Yaskawa INFORM job: tank_top_cylinder_program.JBI

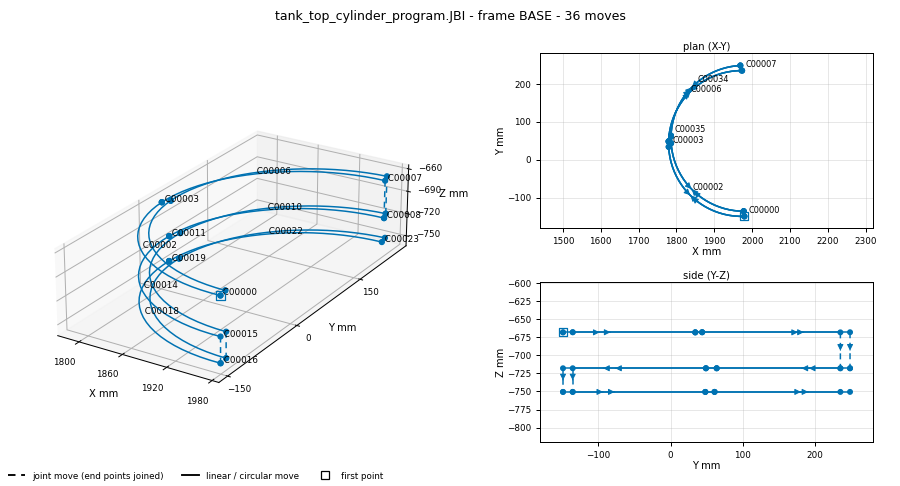
[picture p0: tool path of tank_top_cylinder_program.JBI in frame BASE, 36 of 53 moves have a stored position in this frame; points joined in program order, loops and branches not executed]
/JOB
//NAME tank_top_cylinder_program
//POS
///NPOS 48,0,48,0,0,0
///TOOL 0
///POSTYPE BASE
///RECTAN
///RCONF 0,0,0,0,0,0,0,0,0,0,0,0,0,0,0,0,0,0,0,0,0,0,0,0
C00000=1979.397693,-149.249816,-667.882960,175.000000,-60.000000,92.235388
C00001=1979.397693,-149.249816,-667.882960,175.000000,-60.000000,92.235388
C00002=1833.061579,-90.299080,-667.882960,175.000000,-60.000000,43.881048
C00003=1779.487286,34.344834,-667.882960,175.000000,-60.000000,5.000000
C00004=1779.487286,34.344834,-667.882960,175.000000,-60.000000,5.000000
C00005=1779.487286,34.344834,-667.882960,175.000000,-60.000000,5.000000
C00006=1826.412747,169.432456,-667.882960,-175.000000,-60.000000,-40.948275
C00007=1973.618558,235.799618,-667.882960,-175.000000,-60.000000,-90.515634
C00008=1973.589783,235.799875,-717.744460,175.000000,-60.000000,-90.507073
C00009=1973.589783,235.799875,-717.744460,175.000000,-60.000000,-90.507073
C00010=1835.629981,179.330426,-717.744460,175.000000,-60.000000,-44.972576
C00011=1779.374912,49.143354,-717.744460,-175.000000,-60.000000,-5.000000
C00012=1779.374912,49.143354,-717.744460,-175.000000,-60.000000,-5.000000
C00013=1779.374912,49.143354,-717.744460,-175.000000,-60.000000,-5.000000
C00014=1834.422880,-91.700324,-717.744460,-175.000000,-60.000000,44.462219
C00015=1979.256218,-149.255286,-717.744460,175.000000,-60.000000,92.193270
C00016=1979.223949,-149.256519,-750.568460,175.000000,-60.000000,92.183664
C00017=1979.223949,-149.256519,-750.568460,175.000000,-60.000000,92.183664
C00018=1835.536121,-92.825377,-750.568460,175.000000,-60.000000,44.933056
C00019=1779.350875,48.304771,-750.568460,-175.000000,-60.000000,-5.000000
C00020=1779.350875,48.304771,-750.568460,-175.000000,-60.000000,-5.000000
C00021=1779.350875,48.304771,-750.568460,-175.000000,-60.000000,-5.000000
C00022=1836.839439,180.530381,-750.568460,175.000000,-60.000000,-45.479407
C00023=1971.504480,235.807041,-750.568460,-175.000000,-60.000000,-89.886724
C00024=1977.066518,-135.776203,-667.728960,175.000000,-60.000000,89.707024
C00025=1977.066518,-135.776203,-667.728960,175.000000,-60.000000,89.707024
C00026=1844.462464,-81.919379,-667.728960,175.000000,-60.000000,46.084148
C00027=1785.883314,43.902956,-667.728960,-175.000000,-60.000000,5.000000
C00028=1785.883314,43.902956,-667.728960,-175.000000,-60.000000,5.000000
C00029=1785.883314,43.902956,-667.728960,-175.000000,-60.000000,5.000000
C00030=1833.250365,183.819881,-667.728960,175.000000,-60.000000,-41.252155
C00031=1968.891388,249.207135,-667.728960,175.000000,-60.000000,-87.274035
C00032=1968.707090,249.198272,-717.744960,-175.000000,-60.000000,-87.219146
C00033=1968.707090,249.198272,-717.744960,-175.000000,-60.000000,-87.219146
C00034=1845.123262,196.198971,-717.744960,175.000000,-60.000000,-46.356412
C00035=1785.586247,64.080606,-717.744960,175.000000,-60.000000,-5.000000
C00036=1785.586247,64.080606,-717.744960,175.000000,-60.000000,-5.000000
C00037=1785.586247,64.080606,-717.744960,175.000000,-60.000000,-5.000000
C00038=1834.995615,-72.136289,-717.744960,175.000000,-60.000000,42.033491
C00039=1978.055296,-135.778721,-717.744960,175.000000,-60.000000,90.001169
C00040=1977.931178,-135.778684,-750.538960,-175.000000,-60.000000,89.964246
C00041=1977.931178,-135.778684,-750.538960,-175.000000,-60.000000,89.964246
C00042=1838.032943,-75.427845,-750.538960,175.000000,-60.000000,43.365889
C00043=1785.497479,61.123511,-750.538960,175.000000,-60.000000,-5.000000
C00044=1785.497479,61.123511,-750.538960,175.000000,-60.000000,-5.000000
C00045=1785.497479,61.123511,-750.538960,175.000000,-60.000000,-5.000000
C00046=1842.656575,193.803991,-750.538960,-175.000000,-60.000000,-45.333625
C00047=1968.577731,249.191945,-750.538960,-175.000000,-60.000000,-87.180618
///POSTYPE PULSE
///PULSE
EX00000=93184.0
EX00001=277504.0
///POSTYPE PULSE
///PULSE
EC00000=93184.0
EC00001=93184.0
EC00002=93184.0
EC00003=93184.0
EC00004=93184.0
EC00005=93184.0
EC00006=93184.0
EC00007=93184.0
EC00008=93184.0
EC00009=93184.0
EC00010=93184.0
EC00011=93184.0
EC00012=93184.0
EC00013=93184.0
EC00014=93184.0
EC00015=93184.0
EC00016=93184.0
EC00017=93184.0
EC00018=93184.0
EC00019=93184.0
EC00020=93184.0
EC00021=93184.0
EC00022=93184.0
EC00023=93184.0
EC00024=277504.0
EC00025=277504.0
EC00026=277504.0
EC00027=277504.0
EC00028=277504.0
EC00029=277504.0
EC00030=277504.0
EC00031=277504.0
EC00032=277504.0
EC00033=277504.0
EC00034=277504.0
EC00035=277504.0
EC00036=277504.0
EC00037=277504.0
EC00038=277504.0
EC00039=277504.0
EC00040=277504.0
EC00041=277504.0
EC00042=277504.0
EC00043=277504.0
EC00044=277504.0
EC00045=277504.0
EC00046=277504.0
EC00047=277504.0
//INST
///DATE 2023/08/16 18:11
///ATTR SC,RW,RJ
////FRAME BASE
///GROUP1 RB1,ST1
NOP
MOVJ P009 EX000 VJ=15.00
MOVJ C00000 EC00000 VJ=15.0
CALL JOB:SPYON
MOVC C00001 EC00001 V=150.0
MOVC C00002 EC00002 V=150.0
MOVC C00003 EC00003 V=150.0
MOVJ C00004 EC00004 VJ=15.0
MOVC C00005 EC00005 V=150.0
MOVC C00006 EC00006 V=150.0
MOVC C00007 EC00007 V=150.0
MOVJ C00008 EC00008 VJ=15.0
MOVC C00009 EC00009 V=150.0
MOVC C00010 EC00010 V=150.0
MOVC C00011 EC00011 V=150.0
MOVJ C00012 EC00012 VJ=15.0
MOVC C00013 EC00013 V=150.0
MOVC C00014 EC00014 V=150.0
MOVC C00015 EC00015 V=150.0
MOVJ C00016 EC00016 VJ=15.0
MOVC C00017 EC00017 V=150.0
MOVC C00018 EC00018 V=150.0
MOVC C00019 EC00019 V=150.0
MOVJ C00020 EC00020 VJ=15.0
MOVC C00021 EC00021 V=150.0
MOVC C00022 EC00022 V=150.0
MOVC C00023 EC00023 V=150.0
CALL JOB:SPYOF
MOVJ P009 VJ=15.00
MOVL P009 EX00000 V=150.0
MOVJ C00024 EC00024 VJ=15.0
CALL JOB:SPYON
MOVC C00025 EC00025 V=150.0
MOVC C00026 EC00026 V=150.0
MOVC C00027 EC00027 V=150.0
MOVJ C00028 EC00028 VJ=15.0
MOVC C00029 EC00029 V=150.0
MOVC C00030 EC00030 V=150.0
MOVC C00031 EC00031 V=150.0
MOVJ C00032 EC00032 VJ=15.0
MOVC C00033 EC00033 V=150.0
MOVC C00034 EC00034 V=150.0
MOVC C00035 EC00035 V=150.0
MOVJ C00036 EC00036 VJ=15.0
MOVC C00037 EC00037 V=150.0
MOVC C00038 EC00038 V=150.0
MOVC C00039 EC00039 V=150.0
MOVJ C00040 EC00040 VJ=15.0
MOVC C00041 EC00041 V=150.0
MOVC C00042 EC00042 V=150.0
MOVC C00043 EC00043 V=150.0
MOVJ C00044 EC00044 VJ=15.0
MOVC C00045 EC00045 V=150.0
MOVC C00046 EC00046 V=150.0
MOVC C00047 EC00047 V=150.0
CALL JOB:SPYOF
MOVJ P009 VJ=15.00
MOVL P009 EX00001 V=150.0
END
